% RSLogix 500 project P7.RSS, saved by version 9.00.00.04 %
PROJECT "UNTITLED"    % processor: Bul.1763 MicroLogix 1100 Series B %

PROGRAM FILES
  LAD 2   6 rungs
  LAD 3 "IO"  5 rungs
  LAD 4 "CTRL"  3 rungs
  LAD 5 "CAL"  8 rungs
  LAD 6 "CYCLE"  2 rungs

DATA FILES
  O0 OUTPUT  4 elements
  I1 INPUT  6 elements
  S2 STATUS  66 elements
  B3 BINARY  1 elements
  T4 TIMER  4 elements
  C5 COUNTER  2 elements
  R6 CONTROL  1 elements
  N7 INTEGER  8 elements
  F8 FLOAT  9 elements

LADDER 2
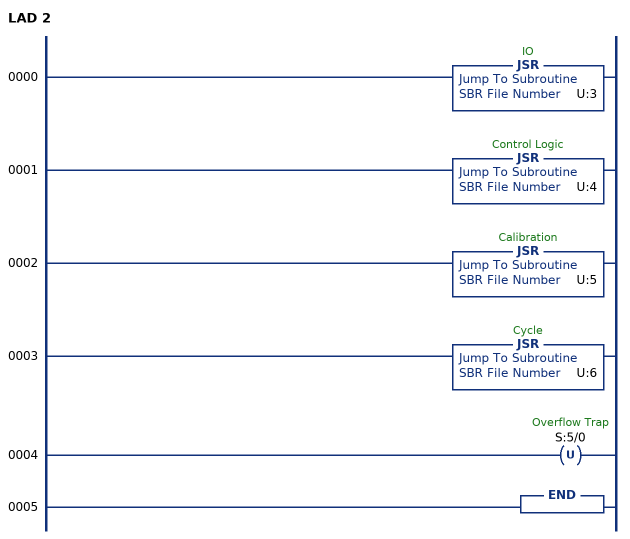
% Rung: 0 %
SOR JSR U:3 EOR
%   U:3  "IO" %
% Rung: 1 %
SOR JSR U:4 EOR
%   U:4  "Control Logic" %
% Rung: 2 %
SOR JSR U:5 EOR
%   U:5  "Calibration" %
% Rung: 3 %
SOR JSR U:6 EOR
%   U:6  "Cycle" %
% Rung: 4 %
SOR OTU S:5/0 EOR
%   S:5/0  "Overflow Trap" %
% Rung: 5 %
SOR END EOR

LADDER 3 "IO"
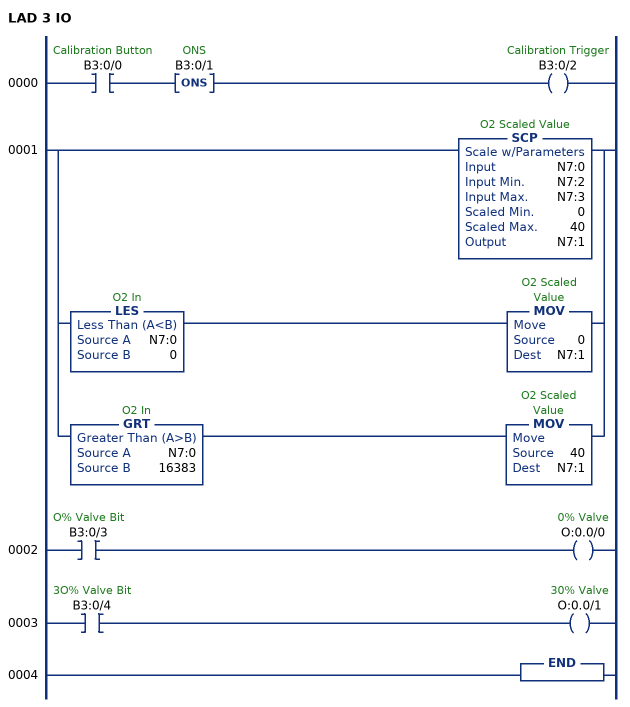
% Rung: 0 %
SOR XIC B3:0/0 ONS B3:0/1 OTE B3:0/2 EOR
%   B3:0/0  "Calibration Button" %
%   B3:0/1  "ONS" %
%   B3:0/2  "Calibration Trigger" %
% Rung: 1 %
SOR BST SCP N7:0 N7:2 N7:3 0 40 N7:1 NXB LES N7:0 0 MOV 0 N7:1 NXB GRT N7:0 16383 MOV 40 N7:1 BND EOR
%   N7:0  "O2 In" %
%   N7:2  "O2 Input Minimum" %
%   N7:3  "O2 Input Maximum" %
%   N7:1  "O2 Scaled Value" %
% Rung: 2 %
SOR XIC B3:0/3 OTE O:0.0/0 EOR
%   B3:0/3  "O% Valve Bit" %
%   O:0.0/0  "0% Valve" %
% Rung: 3 %
SOR XIC B3:0/4 OTE O:0.0/1 EOR
%   B3:0/4  "3O% Valve Bit" %
%   O:0.0/1  "30% Valve" %
% Rung: 4 %
SOR END EOR

LADDER 4 "CTRL"
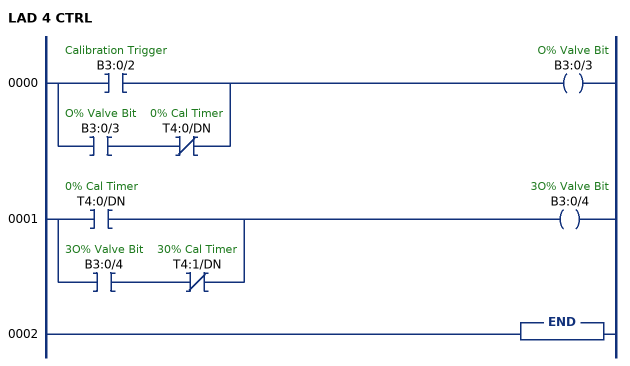
% Rung: 0 %
SOR BST XIC B3:0/2 NXB XIC B3:0/3 XIO T4:0/DN BND OTE B3:0/3 EOR
%   B3:0/2  "Calibration Trigger" %
%   B3:0/3  "O% Valve Bit" %
%   T4:0  "0% Cal Timer" %
% Rung: 1 %
SOR BST XIC T4:0/DN NXB XIC B3:0/4 XIO T4:1/DN BND OTE B3:0/4 EOR
%   T4:0  "0% Cal Timer" %
%   B3:0/4  "3O% Valve Bit" %
%   T4:1  "30% Cal Timer" %
% Rung: 2 %
SOR END EOR

LADDER 5 "CAL"
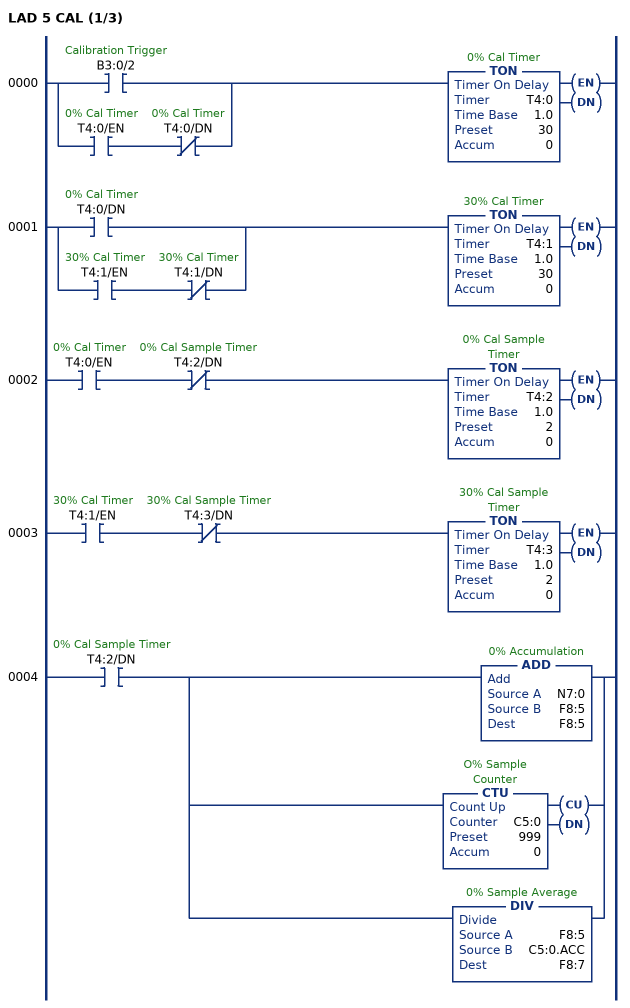
% Rung: 0 %
SOR BST XIC B3:0/2 NXB XIC T4:0/EN XIO T4:0/DN BND TON T4:0 1.0 30 0 EOR
%   B3:0/2  "Calibration Trigger" %
%   T4:0  "0% Cal Timer" %
% Rung: 1 %
SOR BST XIC T4:0/DN NXB XIC T4:1/EN XIO T4:1/DN BND TON T4:1 1.0 30 0 EOR
%   T4:0  "0% Cal Timer" %
%   T4:1  "30% Cal Timer" %
% Rung: 2 %
SOR XIC T4:0/EN XIO T4:2/DN TON T4:2 1.0 2 0 EOR
%   T4:0  "0% Cal Timer" %
%   T4:2  "0% Cal Sample Timer" %
% Rung: 3 %
SOR XIC T4:1/EN XIO T4:3/DN TON T4:3 1.0 2 0 EOR
%   T4:1  "30% Cal Timer" %
%   T4:3  "30% Cal Sample Timer" %
% Rung: 4 %
SOR XIC T4:2/DN BST ADD N7:0 F8:5 F8:5 NXB CTU C5:0 999 0 NXB DIV F8:5 C5:0.ACC F8:7 BND EOR
%   T4:2  "0% Cal Sample Timer" %
%   N7:0  "O2 In" %
%   F8:5  "0% Accumulation" %
%   C5:0  "O% Sample Counter" %
%   F8:7  "0% Sample Average" %

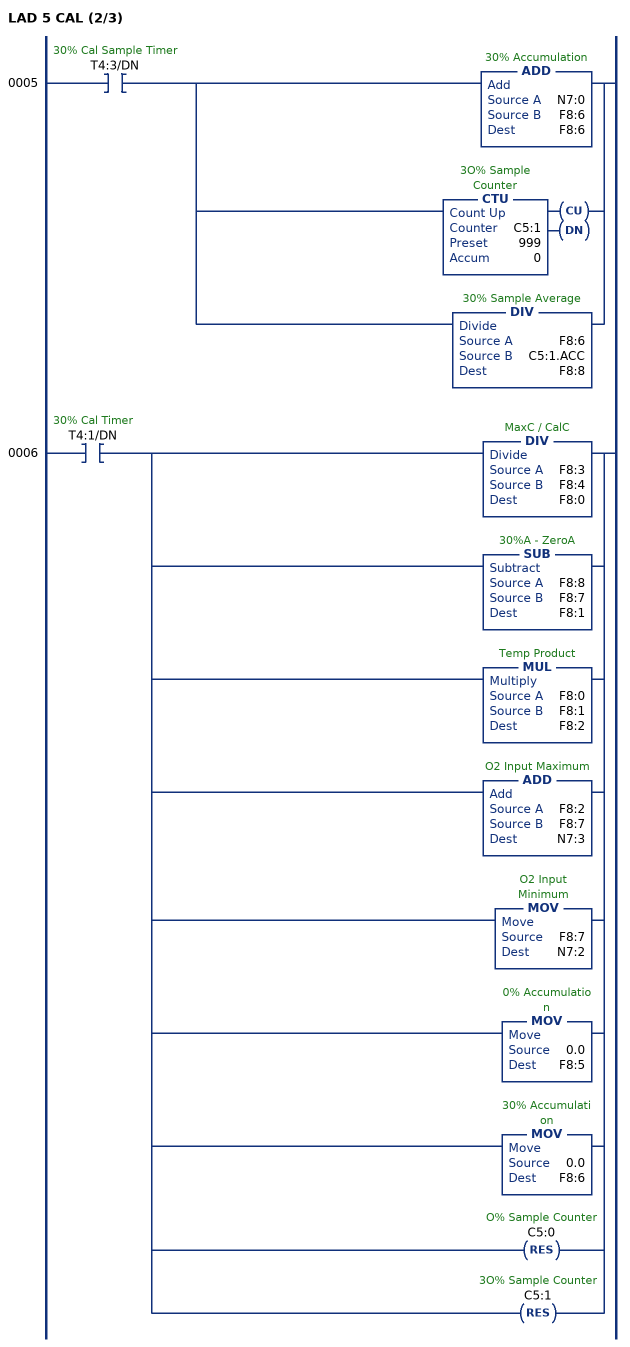
% Rung: 5 %
SOR XIC T4:3/DN BST ADD N7:0 F8:6 F8:6 NXB CTU C5:1 999 0 NXB DIV F8:6 C5:1.ACC F8:8 BND EOR
%   T4:3  "30% Cal Sample Timer" %
%   N7:0  "O2 In" %
%   F8:6  "30% Accumulation" %
%   C5:1  "3O% Sample Counter" %
%   F8:8  "30% Sample Average" %
% Rung: 6 %
SOR XIC T4:1/DN BST DIV F8:3 F8:4 F8:0 NXB SUB F8:8 F8:7 F8:1 NXB MUL F8:0 F8:1 F8:2 NXB ADD F8:2 F8:7 N7:3 NXB MOV F8:7 N7:2 NXB MOV 0.0 F8:5 NXB MOV 0.0 F8:6 NXB RES C5:0 NXB RES C5:1 BND EOR
%   T4:1  "30% Cal Timer" %
%   F8:3  "Max Concentration" %
%   F8:4  "Cal Concentration" %
%   F8:0  "MaxC / CalC" %
%   F8:8  "30% Sample Average" %
%   F8:7  "0% Sample Average" %
%   F8:1  "30%A - ZeroA" %
%   F8:2  "Temp Product" %
%   N7:3  "O2 Input Maximum" %
%   N7:2  "O2 Input Minimum" %
%   F8:5  "0% Accumulation" %
%   F8:6  "30% Accumulation" %
%   C5:0  "O% Sample Counter" %
%   C5:1  "3O% Sample Counter" %

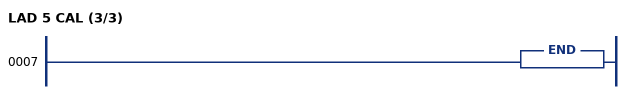
% Rung: 7 %
SOR END EOR

LADDER 6 "CYCLE"
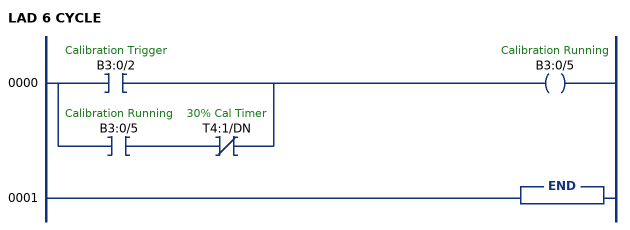
% Rung: 0 %
SOR BST XIC B3:0/2 NXB XIC B3:0/5 XIO T4:1/DN BND OTE B3:0/5 EOR
%   B3:0/2  "Calibration Trigger" %
%   B3:0/5  "Calibration Running" %
%   T4:1  "30% Cal Timer" %
% Rung: 1 %
SOR END EOR

OTHER DOCUMENTED ADDRESSES
  T3  "Cal Sample Timer"

DATA TABLE (non-zero values as saved)
DATA T4
% .PRE .ACC %
% T4:0 % 30 0
% T4:1 % 30 0
% T4:2 % 2 0
% T4:3 % 2 0
DATA C5
% .PRE .ACC %
% C5:0 % 999 0
% C5:1 % 999 0
DATA N7
% N7:0 % 0 0 0 16383 0 0 0 0
DATA F8
% F8:0 % 1.333333 12288 16384 40 30
% F8:5 % 0 184320 0 12288
